// NeuroPLC — Auto-generated IEC 61131-3 SCL
// Graph: mlp | Target: S71200Backend
// Work memory: 75KB | LUT points: 15
// Nodes: 8 | Ops: {'matmul': 4, 'standard_act': 2, 'softmax': 1, 'argmax': 1}


DATA_BLOCK "NeuroPLC_Weights"
{ S7_Optimized_Access := 'FALSE' }
VERSION : 0.1
NON_RETAIN
   STRUCT

   // MatMul 'fc0': W(32×28) + b(32)
   w0 : ARRAY[0..927] OF REAL :=
[0.5694862, -0.0095692, 0.7619486, 0.2215109, -0.3561512, -0.2522623, 0.2582799, 0.0099258
    0.3836571, -0.0658457, 0.1010401, -0.2984352, 0.1934527, -0.2640140, 0.1362384, -0.0190728
    -0.2375232, -0.1084833, -0.3846658, 0.3771667, -0.1136759, -0.1259104, -0.1682155, 0.4097499
    -0.2194012, -0.2356472, -0.1771912, 0.1675407, 0.1454716, -0.3696787, -0.2783369, -0.1873165
    0.0781848, -0.3527579, -0.2131715, -0.4139680, -0.5927966, 0.3198802, -0.5640871, -0.2003005
    0.1832723, 0.2237836, 0.1929916, 0.2185234, 0.1214973, 0.0208249, 0.2776418, 0.6831574
    -0.1655439, -0.2658227, -0.2709237, 0.0986710, 0.1128972, -0.2047481, -0.3872808, 0.1596099
    -0.2523361, 0.2758174, 0.2686562, -0.5177624, -0.1129441, -0.2192100, 0.3343761, -0.0422801
    -0.3068857, 0.2210509, -0.5496964, 0.3709493, 0.0747587, -0.1170707, -0.3195110, 0.0277475
    -0.2577946, 0.0641775, 0.2055912, 0.6039576, -0.5010191, 0.0377836, 0.2038942, -0.0376425
    0.1546009, 0.3260912, -0.1506072, 0.0569262, -0.1928782, -0.1984540, -0.0539345, 0.3094364
    0.2289592, -0.4250050, -0.0399776, 0.0658291, 0.2534966, -0.0973715, -0.3647969, -0.0156060
    -0.5209337, 0.2564455, 0.1338747, 0.3502659, -0.3756513, 0.2530890, 0.0984663, 0.6602526
    0.3365156, -0.2521311, 0.0946512, -0.6085349, -0.5372492, 0.0455726, -0.0786947, 0.0370381
    -0.5858350, -0.7779619, -0.7385424, -0.2071060, 0.2831336, 0.3243212, 0.2366221, -0.2105746
    -0.3834608, -0.6828474, 0.1007835, 0.0381121, 0.3126857, 0.0975034, 0.0499541, -0.0530838
    0.0799674, -0.1505451, -0.4892448, -0.3954702, 0.1594549, 0.2307071, -0.0041823, 0.5944483
    -0.2759206, -0.4257804, -0.3279784, -0.2977980, 0.0038754, 0.3761657, 0.4177073, 0.0741864
    0.3750937, 0.2039272, -0.2429399, -0.3849822, 0.1600508, -0.1581226, -0.0233814, -0.1151747
    -0.5731639, -0.0274457, 0.1195597, -0.2395748, 0.2293357, -0.0251415, 0.3937997, -0.1454628
    -0.0673693, 0.2948158, 0.5630679, -0.3092144, 0.1832785, 0.0043120, 0.0011036, 0.2549984
    0.1242365, -0.1573328, 0.1472307, 0.2971004, 0.1052006, 0.3616425, -0.1347494, -0.3794992
    0.5467421, -0.1476457, 0.3496484, -0.0583753, 0.2853532, -0.3058073, -0.1615329, -0.5229150
    0.2140338, -0.2294949, 0.2921923, 0.0373898, 0.3493846, 0.5938788, 0.0955027, -0.1719695
    0.6582399, -0.4911650, 0.1269870, -0.4129370, -0.2735490, -0.2155660, 0.4269275, -0.1273027
    -0.2414422, -0.3611139, 0.6480063, 0.3808921, -0.2189153, 0.0094489, 0.6784652, 0.3757944
    0.5965886, 0.3704935, 0.3205929, 0.2190031, -0.3913886, 0.2046225, 0.7660633, 0.5648795
    0.0447379, -0.1363681, -0.1653181, -0.3211187, 0.0557173, -0.6775630, 0.2077208, 0.1863764
    0.0122372, -0.1510706, -0.0393031, -0.2373850, 0.3297745, -0.3327326, -0.1183226, 0.3871697
    -0.4481050, -0.2065133, 0.1012533, -0.2578072, 0.0634624, -0.1246978, 0.1465549, -0.5023389
    0.0640146, 0.1963426, 0.6648222, -0.6102669, -0.2871900, -0.3684005, -0.4533643, -0.1819637
    -0.3802012, 0.4682154, 0.1991423, 0.5698866, 0.3063245, 0.1672625, 0.2611240, -0.6845852
    -0.1005014, -0.6641653, -0.2544510, 0.1954752, -0.2994281, 0.3571715, -0.0372742, -0.0310561
    0.1959654, -0.1060541, 0.3827632, -0.3923316, -0.5924090, 0.0670658, 0.3532278, 0.6439264
    0.1193878, -0.5490641, -0.6517076, 0.2266813, 0.2735080, 0.2562127, 0.3711089, -0.0201157
    0.5907255, 0.3026478, 0.0879490, -0.1103418, 0.0830003, 0.0901832, 0.4872787, -0.4248994
    0.6916616, 0.0068263, 0.0377772, -0.3450460, 0.5848706, -0.0756037, 0.0390328, -0.4139087
    -0.1527735, -0.2285863, 0.3310088, 0.2031009, -0.5309294, -0.4607368, 0.1824918, -0.1911459
    -0.1732452, -0.3283744, -0.0425148, -0.0754750, -0.0751830, -0.0057766, -0.0669558, -0.0518108
    -0.1100485, 0.4202482, 0.1722786, 0.2540640, -0.2125306, -0.3108644, -0.1653187, 0.0082027
    0.1613134, 0.5696448, 0.4734836, -0.1820288, -0.0202256, 0.2319008, 0.6178575, -0.1729726
    -0.5705087, -0.4175466, -0.0846097, -0.4305633, -0.0297265, -0.2146564, -0.0228577, 0.4386194
    0.1366172, 0.1275948, 0.2872518, -0.0469490, -0.3430789, -0.2333279, -0.0942715, -0.6695372
    0.3036573, 0.6706407, 0.4867018, 0.2229243, 0.1479198, 0.4786703, -0.1235309, -0.1444162
    -0.1594525, 0.0118241, 0.3302614, 0.4612524, -0.1728074, -0.4940682, 0.2663130, 0.4213447
    0.1559720, 0.0927116, 0.2581408, 0.1484697, 0.5596921, 0.6450443, 0.2316463, -0.3064318
    0.3154030, 0.2504337, 0.2270162, -0.2362736, -0.1822204, 0.7585521, 0.2454521, -0.3572387
    0.1800293, 0.1965537, 0.1946464, 0.1738928, -0.1159788, -0.1791228, 0.3109314, 0.1039406
    -0.2558490, -0.4132357, -0.1826324, -0.0949509, 0.0754630, -0.4951166, -0.0366096, -0.5241205
    0.0701182, 0.5458165, -0.3082272, -0.1620290, 0.2685293, -0.1115321, 0.5528188, 0.1818966
    -0.2705870, -0.4477837, -0.3260813, -0.1751753, 0.3439055, 0.3690660, -0.0775537, -0.3291571
    0.3966570, 0.3747428, 0.2037812, 0.5063270, -0.0363616, -0.0945516, -0.2667596, -0.1880456
    0.2148547, -0.6592890, -0.2238534, -0.2862469, -0.8308039, -0.4430834, -0.0302747, 0.0918460
    -0.3334551, -0.1804388, -0.1097601, 0.3427432, 0.0736062, -0.6790179, -0.2430520, -0.2084594
    0.1491454, -0.0083196, 0.2553293, 0.1678275, 0.0936099, 0.1736043, -0.5376837, -0.4510113
    -0.3174161, 0.2371299, 0.3883051, 0.3464468, 0.1098732, 0.0205052, -0.2641115, -0.3012585
    -0.5463231, -0.0684724, -0.1422806, -0.2644515, -0.4767578, -0.4182616, -0.4673964, -0.0129319
    -0.5374129, -0.1050398, 0.0632549, 0.0568505, 0.2111508, 0.3917949, -0.0330271, 0.2814879
    -0.3214771, 0.3430510, -0.3870021, -0.4042188, 0.1747253, 0.3262924, 0.5594077, 0.0277393
    -0.2604083, 0.0503597, 0.3725081, -0.0544451, 0.0951887, -0.5271522, -0.3720489, 0.0333015
    0.3407656, -0.0524092, -0.3947720, 0.0632993, -0.4918242, -0.0408889, 0.5603451, 0.3429145
    -0.0672607, -0.3218429, -0.3621323, -0.5524946, 0.3105496, 0.3352183, -0.6259544, -0.1107638
    0.0901521, 0.0038500, 0.5420415, 0.2380718, -0.0511688, -0.0771460, -0.0791493, -0.1069665
    0.6399192, -0.0014034, 0.3290343, -0.3565734, 0.2305476, -0.0417552, 0.2942790, -0.1355964
    0.0557771, 0.3271682, -0.3025698, 0.2897500, 0.1278277, -0.1560617, 0.2582703, -0.0549245
    -0.0921321, 0.4996554, 0.0836308, 0.2032579, -0.1741465, -0.2436171, -0.3661414, -0.2924559
    -0.4407195, 0.2304931, -0.2509898, -0.6881460, 0.1500384, 0.4429501, 0.5444623, 0.0644146
    0.1564979, 0.1936211, -0.2217757, 0.1632960, 0.0949209, 0.5449093, 0.3260632, 0.4177442
    -0.1678705, -0.4614883, -0.1780888, 0.0282706, -0.3548764, 0.1119965, -0.6278588, -0.2857478
    0.3291071, -0.2958602, -0.2171935, 0.0488607, -0.2721503, -0.0109805, -0.2872001, -0.3800366
    0.7377275, 0.5175216, 0.4534726, 0.2131705, 0.1694544, 0.1088488, 0.2956495, -0.1219863
    0.4281839, 0.0482728, 0.3261450, 0.0147065, 0.0197347, -0.2837075, -0.2223815, -0.3011971
    0.4010099, 0.3606303, 0.5675586, -0.1933776, 0.1411208, 0.4412328, -0.3157989, 0.0737199
    0.2547267, -0.4104514, 0.3333948, 0.0244799, 0.3485871, -0.1856655, -0.2338329, -0.2214157
    0.4647014, -0.3053385, -0.1758788, -0.2062785, 0.4421045, 0.2903270, 0.2819436, -0.3433319
    -0.0214767, 0.5416198, -0.0143610, -0.1832658, -0.5633022, -0.1308155, 0.1253684, -0.3460040
    -0.0773746, -0.0179889, -0.3036036, 0.0990553, -0.2073587, 0.0275394, 0.0471204, -0.0187443
    0.4038751, 0.0922068, -0.2135524, -0.4082574, -0.0358560, -0.1610684, -0.4163499, 0.2467240
    0.0747931, 0.3987921, 0.1632655, -0.3848493, 0.1649167, -0.6442378, -0.4510081, -0.2822698
    0.4664556, -0.2991767, -0.0362801, -0.3327457, -0.3074295, 0.1606831, -0.0541677, -0.5748461
    0.3949239, -0.2336025, -0.0525538, 0.3131756, -0.0032524, -0.0003879, 0.3644529, 0.3278647
    -0.0496909, -0.0200011, 0.4739185, -0.3886660, 0.0855980, -0.4665208, 0.4008028, -0.5448800
    -0.4093939, -0.1329360, 0.2988919, -0.0788539, 0.0282110, -0.1015701, 0.5736219, -0.2615215
    0.0237927, 0.0321014, -0.1239056, -0.2004481, -0.0194097, -0.1323835, -0.0777957, 0.0366594
    0.1079154, 0.4157223, -0.2902254, 0.4283061, 0.0650300, 0.1249261, -0.2917063, -0.1270394
    0.0782463, 0.5982807, 0.1017760, 0.1843081, -0.6125457, 0.2722199, -0.0728571, -0.5004624
    0.4432183, 0.4912130, 0.0002442, -0.0942999, 0.5940161, -0.1235101, 0.3478113, 0.0345737
    -0.0406947, 0.6151400, 0.2030335, -0.3236780, -0.6019017, -0.4779230, -0.8101817, -0.2094196
    -0.3149875, 0.3055148, -0.2818980, 0.2800311, -0.8234739, -0.6584272, 0.2585062, 0.0584044
    -0.5591815, -0.0547792, 0.0355113, 0.2701355, -0.5936313, 0.3193162, 0.1195579, 0.0537417
    0.6140408, 0.5008627, -0.0104372, 0.2329175, -0.0168664, 0.0332739, 0.3730388, 0.1635417
    0.7335413, 0.5691491, 0.0170918, 0.2825087, 0.0198349, 0.4498756, 0.4100120, -0.2479021
    0.2850291, -0.1702987, -0.4980538, -0.0941117, 0.4272463, -0.2824812, 0.6535753, 0.2375765
    0.4509313, -0.0013205, 0.1127060, -0.1239916, 0.3028973, 0.0927592, -0.3168923, 0.1611173
    0.4917028, 0.0417323, 0.3917417, -0.0557213, -0.2345485, 0.3833969, 0.3747815, -0.1519468
    -0.3892233, -0.0699942, -0.3351573, -0.3026012, -0.1781991, 0.4689204, -0.1804391, -0.2284776
    -0.3932275, 0.2445571, -0.1087966, -0.2825441, -0.2301650, 0.5091258, -0.7006359, 0.0339814
    0.1417895, 0.1839303, 0.2910166, 0.1044962, 0.0580844, 0.6158280, -0.0284938, 0.0542879
    0.1680317, 0.2264472, -0.2030084, 0.0756811, -0.2188872, -0.2264328, -0.1813061, -0.2645762
    0.4621922, -0.4514092, 0.3058094, 0.3434274, 0.3808913, -0.3231871, 0.2469297, -0.1890893
    0.0499585, -0.3218643, 0.6025205, 0.0650566, -0.2298092, 0.5071256, -0.2657916, -0.1830709
    0.0415640, -0.1594847, -0.0321660, -0.0346579, -0.3819390, 0.2074234, 0.3919429, 0.0324158
    -0.0215873, -0.1329270, 0.0735578, 0.3148956, -0.4435450, -0.3320747, -0.1767979, -0.4104172
    0.3253109, -0.1773608, -0.4930988, 0.3281353, 0.3916833, -0.1541856, 0.1263307, 0.0426248
    -0.5533415, 0.0726361, -0.4881184, -0.1073755, -0.5946367, -0.5742470, 0.1233901, -0.0872265
    0.2010813, 0.4012275, 0.3290967, 0.3005436, -0.0111396, -0.4794478, -0.0532993, -0.1733176
    -0.1260332, 0.1089438, 0.0391418, -0.2468968, 0.4689822, -0.4640872, 0.2532913, -0.2343228
    0.2661497, -0.4386278, 0.0468966, -0.3265733, -0.1916417, 0.5178355, 0.2822486, -0.1077720
    0.3286300, -0.0029810, -0.3535745, -0.1011055, 0.1318278, 0.0674391, 0.0591611, -0.1122496
    0.4686061, -0.4002847, 0.0749937, -0.1933431, 0.2702274, -0.1278288, -0.1761822, -0.2737747
    0.4466998, 0.0271071, 0.1916832, 0.4834492, 0.0259246, -0.4892190, 0.2059345, -0.0822330
    -0.4142632, 0.5404200, -0.1093403, 0.0186543, 0.6250578, -0.2241697, 0.3088920, 0.1112378
    -0.1609981, -0.0371174, 0.0221225, 0.0337845, 0.2616802, 0.1264098, 0.1833381, 0.1271529
    0.0488858, 0.0241906, -0.3121075, 0.0973287, -0.0882614, -0.3344531, -0.1306882, 0.1518650
    0.0104939, -0.0685202, -0.0953050, 0.0008646, 0.2513834, 0.0002911, 0.1923783, 0.1726166
    0.3154603, 0.0885571, 0.0390019, 0.0755870, 0.1380671, 0.1447226, 0.0485010, 0.1450995];

   // MatMul 'fc1': W(16×32) + b(16)
   w1 : ARRAY[0..527] OF REAL :=
[0.3448875, -0.0985299, -0.2385274, 0.1068773, 0.5171419, -0.1054032, 0.2936411, -0.4853331
    -0.3005029, 0.2366145, 0.3783182, 0.1278910, 0.0211917, -0.1069832, -0.2683547, -0.0976455
    0.6765909, 0.5036446, 0.3599868, 0.0810751, -0.0792580, -0.2718676, -0.4316851, -0.1867653
    0.2037492, -0.0189868, -0.0119788, 0.3331117, -0.1736732, -0.4839838, -0.0297980, -0.6352752
    0.4027197, -0.5263022, 0.2703936, 0.1180763, -0.3752257, -0.6156019, -0.4087748, 0.1517635
    0.2814839, -0.3188637, 0.4876765, 0.1747880, -0.1799005, -0.3207765, 0.6545156, -0.3893254
    -0.3369366, -0.4376430, 0.0413780, -0.1731163, 0.3791941, 0.0461393, 0.0816816, 0.3956819
    -0.3843228, -0.7061806, -0.6190179, -0.4308152, 0.2132129, 0.4490756, -0.2397823, 0.3091693
    -0.1736172, -0.6044765, 0.2081352, 0.4768652, -0.2759739, 0.1133698, -0.0100859, -0.6772556
    0.5169631, 0.1017481, -0.0672581, -0.4697476, -0.1098660, -0.1401970, -0.4618214, -0.2387714
    -0.3492894, -0.2289385, 0.3859353, 0.3484918, 0.0570800, 0.4838708, 0.4412340, 0.1156965
    0.4213234, -0.2558614, 0.2997079, -0.0041088, -0.2610477, -0.2681805, 0.7025032, 0.4033620
    0.0018223, 0.3965206, -0.1132530, 0.3405365, 0.4333419, 0.0468351, -0.4313038, -0.5938676
    -0.1057017, 0.3874305, -0.3047897, -0.3605830, -0.0865778, 0.0169620, -0.2818013, -0.2056310
    0.2889744, -0.2389124, -0.5219849, -0.5379763, -0.3595321, 0.2131797, 0.2746126, 0.2555465
    -0.3816569, -0.1742714, -0.3458711, -0.4732965, 0.3816739, 0.4522255, 0.4340182, 0.1317699
    0.0887004, -0.1704083, 0.2312619, -0.1512796, 0.1522121, -0.3580639, 0.3120518, -0.0891345
    -0.5189782, 0.6759704, 0.8410841, -0.4388631, 0.3120123, 0.0530660, -0.1540236, -0.1420563
    0.3882907, 0.3881267, 0.4476533, 0.4830106, 0.2335594, 0.1241002, -0.2032309, -0.5769788
    0.3601961, 0.5940281, -0.3626602, 0.1981693, -0.0685700, -0.0704796, 0.0195035, -0.4674689
    -0.2348353, -0.3250483, 0.1978887, -0.0533809, 0.5541837, 0.0647560, 0.1574209, -0.4176951
    -0.0328900, -0.4697271, -0.0496295, -0.1912494, -0.2456453, -0.3518490, 0.0067706, 0.6691334
    0.5995317, 0.3372136, -0.2781896, 0.2096184, -0.4983254, -0.0787928, -0.2063265, -0.2567849
    -0.2985751, 0.2627156, 0.1459312, 0.4578165, 0.0136775, 0.4329558, -0.2819005, 0.0772760
    0.1485205, 0.0424627, -0.5533946, -0.3114872, -0.0971009, 0.1043289, -0.0080725, 0.0561389
    0.1712011, -0.2093053, -0.4844932, 0.5200891, -0.4811763, -0.2097965, -0.1644997, 0.0035760
    0.2773729, 0.4809147, -0.3132524, -0.0345517, 0.5111094, 0.1451371, 0.0575851, 0.1672285
    0.3724994, 0.0500904, -0.0895519, 0.0279228, -0.0756062, -0.6023685, 0.5966649, -0.4288191
    -0.2491551, 0.1842164, 0.1995990, 0.3348442, -0.6874152, 0.0923893, 0.5566139, 0.6076588
    0.4055642, 0.1035502, -0.2282035, 0.0315236, 0.3474000, 0.1027276, 0.0550077, -0.1958367
    -0.1637788, 0.2277053, -0.1716563, 0.1922517, 0.2188656, 0.0905953, -0.2237651, 0.4562837
    -0.4297628, 0.0540233, -0.2155596, -0.4905677, 0.2578664, -0.0752592, 0.3203000, 0.2922962
    0.6623323, -0.2237271, -0.3789170, -0.3014932, 0.3499548, -0.3618023, -0.1381309, -0.2487616
    -0.2042618, -0.3798007, 0.2168026, -0.5617495, 0.5470159, 0.3855161, -0.1744407, -0.0063227
    -0.0175713, 0.4657946, 0.2311470, 0.2995405, -0.2337339, 0.2714463, -0.1801859, -0.2387183
    0.2680195, 0.4208193, 0.0763752, -0.0259924, -0.5796329, -0.4459113, -0.0650182, 0.0992380
    -0.2287219, 0.1592736, 0.2655782, -0.7133095, -0.0750051, 0.1930008, 0.2515846, -0.1046810
    0.3638516, -0.5185701, -0.1378490, 0.1176404, -0.1728815, -0.4648141, -0.0106897, 0.2669196
    -0.2057847, -0.0459625, -0.0872513, -0.5442434, 0.4806913, -0.2794292, 0.6181495, 0.4071167
    -0.3071254, 0.1203253, 0.3505305, -0.5886531, -0.2951987, 0.3731146, 0.2878209, 0.2473200
    -0.1784255, 0.4152616, 0.5053530, 0.2126275, 0.3228098, -0.3918779, -0.1658438, 0.5003296
    -0.0053924, 0.0667791, 0.4097935, 0.1006095, 0.6046916, -0.0676274, -0.1915504, 0.3883604
    0.4911340, 0.5468511, -0.1983627, -0.0676885, -0.3710055, 0.1606412, 0.4564988, -0.5501073
    -0.1039538, -0.0296496, -0.5341417, -0.2000433, 0.2511403, 0.3043574, -0.1509714, 0.4652316
    0.5162573, -0.4559039, 0.1557730, -0.3858083, 0.0727105, -0.4605626, -0.0643399, -0.2012528
    -0.2376907, 0.6337410, 0.7189264, 0.2091954, 0.7626936, 0.3527288, -0.1358239, 0.3472250
    -0.0854939, 0.3039412, 0.2409862, 0.4435183, 0.4328762, -0.0231600, -0.1171540, 0.0108573
    -0.0911193, -0.5950353, -0.1391228, 0.1307337, -0.1149503, -0.0330209, -0.4081971, -0.3619282
    -0.1067709, -0.0438268, 0.1861137, 0.1071503, -0.6722144, 0.5858943, 0.1327110, 0.3459137
    0.3487434, 0.0373104, -0.2565190, 0.4223759, -0.2403768, -0.0137525, 0.1307058, -0.5750338
    -0.6017820, 0.1216069, -0.0930582, 0.0528917, 0.2642088, 0.1213500, -0.0773624, 0.1509228
    0.1637788, -0.0275139, 0.5865979, -0.2206961, 0.5099282, 0.2631257, 0.4237445, 0.4448525
    0.4446503, 0.0053865, -0.5579309, -0.1395655, -0.1579983, -0.3564516, 0.0891758, 0.1217025
    -0.3250042, -0.0731721, 0.5731527, 0.3349074, -0.2764013, 0.3669565, 0.1658501, -0.0952915
    0.1848216, -0.3777516, 0.4125981, -0.2243889, 0.2011978, 0.3032005, 0.0724154, 0.2386405
    -0.4659944, -0.5817581, -0.3680228, -0.5429725, -0.4282436, -0.0057439, 0.1407171, -0.0961595
    -0.0304086, -0.5598830, -0.5288109, 0.2501028, -0.1907448, 0.3364898, 0.3753116, -0.1153062
    -0.0149126, -0.3870158, -0.1154010, 0.0744122, -0.4487402, -0.2563244, 0.0335258, -0.1682583
    0.0443628, 0.3070406, -0.0503107, 0.0992935, 0.5251856, 0.6111719, 0.6419194, 0.1297791
    0.1860752, -0.1274762, 0.3434472, 0.5505610, 0.3397494, -0.5685602, 0.0005795, -0.1080624
    0.3114881, 0.4475129, 0.1615055, -0.4390773, -0.0133804, -0.3265319, -0.5983120, -0.2533576
    0.2004646, -0.2516977, -0.2211783, -0.0643062, 0.1233937, 0.1260124, -0.2689813, 0.3791626
    0.3063162, -0.2886556, -0.1805890, -0.1727612, -0.2364416, -0.0335479, 0.1661869, 0.1447821
    -0.1905543, -0.4342808, -0.0012427, -0.4948293, 0.0922625, 0.0781584, 0.4070034, 0.0575855
    -0.0313972, -0.1867536, 0.2673712, 0.0710777, -0.2155338, 0.0103840, 0.4061291, -0.0612305
    0.0899094, 0.1921517, 0.1069144, -0.0515455, 0.1089574, -0.1325741, 0.2726102, 0.1574048];

   // MatMul 'fc2': W(4×16) + b(4)
   w2 : ARRAY[0..67] OF REAL :=
[-0.0865753, -0.5062438, 0.1554476, 0.7071172, -0.1023560, 0.5811852, -0.6674285, -0.6164539
    -0.8109480, 0.6379222, 0.3449526, -0.0613255, -0.0052660, -0.7050505, -0.6678494, 0.7979829
    -0.0429653, -0.3721911, 0.9616893, -0.2787606, -0.1421925, -0.1321686, 0.1806948, -0.1417111
    -0.4919258, 0.7062184, -0.4885310, -0.5391713, 0.7159519, -0.5416421, 0.8190475, -0.2587632
    0.7209747, -0.5606546, 0.2996863, -0.4360698, 0.6557293, 0.7114502, -0.0711865, -0.5944882
    0.5009670, -0.2733661, 0.0057439, 0.7727029, -0.5340657, 0.0551448, 0.2726173, -0.4893947
    0.2866370, 0.6904863, -0.7133542, 0.1576146, 0.5721015, 0.0582882, -0.7719719, 0.2141585
    -0.2926230, -0.4390040, 0.2077623, 0.5338089, 0.5839869, 0.7652564, -0.3743652, -0.1907377
    -0.1430807, 0.2929625, 0.1342851, -0.1236853];

   // Total: 3 array blocks
   END_STRUCT;
BEGIN
END_DATA_BLOCK

FUNCTION_BLOCK "NeuroPLC_Inference"
{ S7_Optimized_Access := 'FALSE' }
VERSION : 0.1
VAR_INPUT
    features : ARRAY[0..27] OF REAL;
END_VAR

VAR_OUTPUT
    fault_class : INT;
    confidence : REAL;
END_VAR

VAR
    i, j, k : INT;
    sum_val, max_val, t_val : REAL;
    v0 : ARRAY[0..27] OF REAL;
    v1 : ARRAY[0..31] OF REAL;
    v2 : ARRAY[0..31] OF REAL;
    v3 : ARRAY[0..15] OF REAL;
    v4 : ARRAY[0..15] OF REAL;
    v5 : ARRAY[0..3] OF REAL;
    v6 : ARRAY[0..3] OF REAL;
END_VAR

BEGIN
    // ---- Input ----
    FOR i := 0 TO 27 DO
        v0[i] := features[i];
    END_FOR;

    // ---- fc0: MatMul(28→32) ----
    // W = "NeuroPLC_Weights".w0[:896],   b = w0[896:]
    v1[0] := "NeuroPLC_Weights".w0[896 + 0];
    FOR i := 0 TO 27 DO
        v1[0] := v1[0] + "NeuroPLC_Weights".w0[0 + i] * v0[i];
    END_FOR;
    v1[1] := "NeuroPLC_Weights".w0[896 + 1];
    FOR i := 0 TO 27 DO
        v1[1] := v1[1] + "NeuroPLC_Weights".w0[28 + i] * v0[i];
    END_FOR;
    v1[2] := "NeuroPLC_Weights".w0[896 + 2];
    FOR i := 0 TO 27 DO
        v1[2] := v1[2] + "NeuroPLC_Weights".w0[56 + i] * v0[i];
    END_FOR;
    v1[3] := "NeuroPLC_Weights".w0[896 + 3];
    FOR i := 0 TO 27 DO
        v1[3] := v1[3] + "NeuroPLC_Weights".w0[84 + i] * v0[i];
    END_FOR;
    v1[4] := "NeuroPLC_Weights".w0[896 + 4];
    FOR i := 0 TO 27 DO
        v1[4] := v1[4] + "NeuroPLC_Weights".w0[112 + i] * v0[i];
    END_FOR;
    v1[5] := "NeuroPLC_Weights".w0[896 + 5];
    FOR i := 0 TO 27 DO
        v1[5] := v1[5] + "NeuroPLC_Weights".w0[140 + i] * v0[i];
    END_FOR;
    v1[6] := "NeuroPLC_Weights".w0[896 + 6];
    FOR i := 0 TO 27 DO
        v1[6] := v1[6] + "NeuroPLC_Weights".w0[168 + i] * v0[i];
    END_FOR;
    v1[7] := "NeuroPLC_Weights".w0[896 + 7];
    FOR i := 0 TO 27 DO
        v1[7] := v1[7] + "NeuroPLC_Weights".w0[196 + i] * v0[i];
    END_FOR;
    v1[8] := "NeuroPLC_Weights".w0[896 + 8];
    FOR i := 0 TO 27 DO
        v1[8] := v1[8] + "NeuroPLC_Weights".w0[224 + i] * v0[i];
    END_FOR;
    v1[9] := "NeuroPLC_Weights".w0[896 + 9];
    FOR i := 0 TO 27 DO
        v1[9] := v1[9] + "NeuroPLC_Weights".w0[252 + i] * v0[i];
    END_FOR;
    v1[10] := "NeuroPLC_Weights".w0[896 + 10];
    FOR i := 0 TO 27 DO
        v1[10] := v1[10] + "NeuroPLC_Weights".w0[280 + i] * v0[i];
    END_FOR;
    v1[11] := "NeuroPLC_Weights".w0[896 + 11];
    FOR i := 0 TO 27 DO
        v1[11] := v1[11] + "NeuroPLC_Weights".w0[308 + i] * v0[i];
    END_FOR;
    v1[12] := "NeuroPLC_Weights".w0[896 + 12];
    FOR i := 0 TO 27 DO
        v1[12] := v1[12] + "NeuroPLC_Weights".w0[336 + i] * v0[i];
    END_FOR;
    v1[13] := "NeuroPLC_Weights".w0[896 + 13];
    FOR i := 0 TO 27 DO
        v1[13] := v1[13] + "NeuroPLC_Weights".w0[364 + i] * v0[i];
    END_FOR;
    v1[14] := "NeuroPLC_Weights".w0[896 + 14];
    FOR i := 0 TO 27 DO
        v1[14] := v1[14] + "NeuroPLC_Weights".w0[392 + i] * v0[i];
    END_FOR;
    v1[15] := "NeuroPLC_Weights".w0[896 + 15];
    FOR i := 0 TO 27 DO
        v1[15] := v1[15] + "NeuroPLC_Weights".w0[420 + i] * v0[i];
    END_FOR;
    v1[16] := "NeuroPLC_Weights".w0[896 + 16];
    FOR i := 0 TO 27 DO
        v1[16] := v1[16] + "NeuroPLC_Weights".w0[448 + i] * v0[i];
    END_FOR;
    v1[17] := "NeuroPLC_Weights".w0[896 + 17];
    FOR i := 0 TO 27 DO
        v1[17] := v1[17] + "NeuroPLC_Weights".w0[476 + i] * v0[i];
    END_FOR;
    v1[18] := "NeuroPLC_Weights".w0[896 + 18];
    FOR i := 0 TO 27 DO
        v1[18] := v1[18] + "NeuroPLC_Weights".w0[504 + i] * v0[i];
    END_FOR;
    v1[19] := "NeuroPLC_Weights".w0[896 + 19];
    FOR i := 0 TO 27 DO
        v1[19] := v1[19] + "NeuroPLC_Weights".w0[532 + i] * v0[i];
    END_FOR;
    v1[20] := "NeuroPLC_Weights".w0[896 + 20];
    FOR i := 0 TO 27 DO
        v1[20] := v1[20] + "NeuroPLC_Weights".w0[560 + i] * v0[i];
    END_FOR;
    v1[21] := "NeuroPLC_Weights".w0[896 + 21];
    FOR i := 0 TO 27 DO
        v1[21] := v1[21] + "NeuroPLC_Weights".w0[588 + i] * v0[i];
    END_FOR;
    v1[22] := "NeuroPLC_Weights".w0[896 + 22];
    FOR i := 0 TO 27 DO
        v1[22] := v1[22] + "NeuroPLC_Weights".w0[616 + i] * v0[i];
    END_FOR;
    v1[23] := "NeuroPLC_Weights".w0[896 + 23];
    FOR i := 0 TO 27 DO
        v1[23] := v1[23] + "NeuroPLC_Weights".w0[644 + i] * v0[i];
    END_FOR;
    v1[24] := "NeuroPLC_Weights".w0[896 + 24];
    FOR i := 0 TO 27 DO
        v1[24] := v1[24] + "NeuroPLC_Weights".w0[672 + i] * v0[i];
    END_FOR;
    v1[25] := "NeuroPLC_Weights".w0[896 + 25];
    FOR i := 0 TO 27 DO
        v1[25] := v1[25] + "NeuroPLC_Weights".w0[700 + i] * v0[i];
    END_FOR;
    v1[26] := "NeuroPLC_Weights".w0[896 + 26];
    FOR i := 0 TO 27 DO
        v1[26] := v1[26] + "NeuroPLC_Weights".w0[728 + i] * v0[i];
    END_FOR;
    v1[27] := "NeuroPLC_Weights".w0[896 + 27];
    FOR i := 0 TO 27 DO
        v1[27] := v1[27] + "NeuroPLC_Weights".w0[756 + i] * v0[i];
    END_FOR;
    v1[28] := "NeuroPLC_Weights".w0[896 + 28];
    FOR i := 0 TO 27 DO
        v1[28] := v1[28] + "NeuroPLC_Weights".w0[784 + i] * v0[i];
    END_FOR;
    v1[29] := "NeuroPLC_Weights".w0[896 + 29];
    FOR i := 0 TO 27 DO
        v1[29] := v1[29] + "NeuroPLC_Weights".w0[812 + i] * v0[i];
    END_FOR;
    v1[30] := "NeuroPLC_Weights".w0[896 + 30];
    FOR i := 0 TO 27 DO
        v1[30] := v1[30] + "NeuroPLC_Weights".w0[840 + i] * v0[i];
    END_FOR;
    v1[31] := "NeuroPLC_Weights".w0[896 + 31];
    FOR i := 0 TO 27 DO
        v1[31] := v1[31] + "NeuroPLC_Weights".w0[868 + i] * v0[i];
    END_FOR;

    // ---- relu0: RELU ----
    IF v1[0] > 0.0 THEN v2[0] := v1[0]; ELSE v2[0] := 0.0; END_IF;
    IF v1[1] > 0.0 THEN v2[1] := v1[1]; ELSE v2[1] := 0.0; END_IF;
    IF v1[2] > 0.0 THEN v2[2] := v1[2]; ELSE v2[2] := 0.0; END_IF;
    IF v1[3] > 0.0 THEN v2[3] := v1[3]; ELSE v2[3] := 0.0; END_IF;
    IF v1[4] > 0.0 THEN v2[4] := v1[4]; ELSE v2[4] := 0.0; END_IF;
    IF v1[5] > 0.0 THEN v2[5] := v1[5]; ELSE v2[5] := 0.0; END_IF;
    IF v1[6] > 0.0 THEN v2[6] := v1[6]; ELSE v2[6] := 0.0; END_IF;
    IF v1[7] > 0.0 THEN v2[7] := v1[7]; ELSE v2[7] := 0.0; END_IF;
    IF v1[8] > 0.0 THEN v2[8] := v1[8]; ELSE v2[8] := 0.0; END_IF;
    IF v1[9] > 0.0 THEN v2[9] := v1[9]; ELSE v2[9] := 0.0; END_IF;
    IF v1[10] > 0.0 THEN v2[10] := v1[10]; ELSE v2[10] := 0.0; END_IF;
    IF v1[11] > 0.0 THEN v2[11] := v1[11]; ELSE v2[11] := 0.0; END_IF;
    IF v1[12] > 0.0 THEN v2[12] := v1[12]; ELSE v2[12] := 0.0; END_IF;
    IF v1[13] > 0.0 THEN v2[13] := v1[13]; ELSE v2[13] := 0.0; END_IF;
    IF v1[14] > 0.0 THEN v2[14] := v1[14]; ELSE v2[14] := 0.0; END_IF;
    IF v1[15] > 0.0 THEN v2[15] := v1[15]; ELSE v2[15] := 0.0; END_IF;
    IF v1[16] > 0.0 THEN v2[16] := v1[16]; ELSE v2[16] := 0.0; END_IF;
    IF v1[17] > 0.0 THEN v2[17] := v1[17]; ELSE v2[17] := 0.0; END_IF;
    IF v1[18] > 0.0 THEN v2[18] := v1[18]; ELSE v2[18] := 0.0; END_IF;
    IF v1[19] > 0.0 THEN v2[19] := v1[19]; ELSE v2[19] := 0.0; END_IF;
    IF v1[20] > 0.0 THEN v2[20] := v1[20]; ELSE v2[20] := 0.0; END_IF;
    IF v1[21] > 0.0 THEN v2[21] := v1[21]; ELSE v2[21] := 0.0; END_IF;
    IF v1[22] > 0.0 THEN v2[22] := v1[22]; ELSE v2[22] := 0.0; END_IF;
    IF v1[23] > 0.0 THEN v2[23] := v1[23]; ELSE v2[23] := 0.0; END_IF;
    IF v1[24] > 0.0 THEN v2[24] := v1[24]; ELSE v2[24] := 0.0; END_IF;
    IF v1[25] > 0.0 THEN v2[25] := v1[25]; ELSE v2[25] := 0.0; END_IF;
    IF v1[26] > 0.0 THEN v2[26] := v1[26]; ELSE v2[26] := 0.0; END_IF;
    IF v1[27] > 0.0 THEN v2[27] := v1[27]; ELSE v2[27] := 0.0; END_IF;
    IF v1[28] > 0.0 THEN v2[28] := v1[28]; ELSE v2[28] := 0.0; END_IF;
    IF v1[29] > 0.0 THEN v2[29] := v1[29]; ELSE v2[29] := 0.0; END_IF;
    IF v1[30] > 0.0 THEN v2[30] := v1[30]; ELSE v2[30] := 0.0; END_IF;
    IF v1[31] > 0.0 THEN v2[31] := v1[31]; ELSE v2[31] := 0.0; END_IF;

    // ---- fc1: MatMul(32→16) ----
    // W = "NeuroPLC_Weights".w1[:512],   b = w1[512:]
    v3[0] := "NeuroPLC_Weights".w1[512 + 0];
    FOR i := 0 TO 31 DO
        v3[0] := v3[0] + "NeuroPLC_Weights".w1[0 + i] * v2[i];
    END_FOR;
    v3[1] := "NeuroPLC_Weights".w1[512 + 1];
    FOR i := 0 TO 31 DO
        v3[1] := v3[1] + "NeuroPLC_Weights".w1[32 + i] * v2[i];
    END_FOR;
    v3[2] := "NeuroPLC_Weights".w1[512 + 2];
    FOR i := 0 TO 31 DO
        v3[2] := v3[2] + "NeuroPLC_Weights".w1[64 + i] * v2[i];
    END_FOR;
    v3[3] := "NeuroPLC_Weights".w1[512 + 3];
    FOR i := 0 TO 31 DO
        v3[3] := v3[3] + "NeuroPLC_Weights".w1[96 + i] * v2[i];
    END_FOR;
    v3[4] := "NeuroPLC_Weights".w1[512 + 4];
    FOR i := 0 TO 31 DO
        v3[4] := v3[4] + "NeuroPLC_Weights".w1[128 + i] * v2[i];
    END_FOR;
    v3[5] := "NeuroPLC_Weights".w1[512 + 5];
    FOR i := 0 TO 31 DO
        v3[5] := v3[5] + "NeuroPLC_Weights".w1[160 + i] * v2[i];
    END_FOR;
    v3[6] := "NeuroPLC_Weights".w1[512 + 6];
    FOR i := 0 TO 31 DO
        v3[6] := v3[6] + "NeuroPLC_Weights".w1[192 + i] * v2[i];
    END_FOR;
    v3[7] := "NeuroPLC_Weights".w1[512 + 7];
    FOR i := 0 TO 31 DO
        v3[7] := v3[7] + "NeuroPLC_Weights".w1[224 + i] * v2[i];
    END_FOR;
    v3[8] := "NeuroPLC_Weights".w1[512 + 8];
    FOR i := 0 TO 31 DO
        v3[8] := v3[8] + "NeuroPLC_Weights".w1[256 + i] * v2[i];
    END_FOR;
    v3[9] := "NeuroPLC_Weights".w1[512 + 9];
    FOR i := 0 TO 31 DO
        v3[9] := v3[9] + "NeuroPLC_Weights".w1[288 + i] * v2[i];
    END_FOR;
    v3[10] := "NeuroPLC_Weights".w1[512 + 10];
    FOR i := 0 TO 31 DO
        v3[10] := v3[10] + "NeuroPLC_Weights".w1[320 + i] * v2[i];
    END_FOR;
    v3[11] := "NeuroPLC_Weights".w1[512 + 11];
    FOR i := 0 TO 31 DO
        v3[11] := v3[11] + "NeuroPLC_Weights".w1[352 + i] * v2[i];
    END_FOR;
    v3[12] := "NeuroPLC_Weights".w1[512 + 12];
    FOR i := 0 TO 31 DO
        v3[12] := v3[12] + "NeuroPLC_Weights".w1[384 + i] * v2[i];
    END_FOR;
    v3[13] := "NeuroPLC_Weights".w1[512 + 13];
    FOR i := 0 TO 31 DO
        v3[13] := v3[13] + "NeuroPLC_Weights".w1[416 + i] * v2[i];
    END_FOR;
    v3[14] := "NeuroPLC_Weights".w1[512 + 14];
    FOR i := 0 TO 31 DO
        v3[14] := v3[14] + "NeuroPLC_Weights".w1[448 + i] * v2[i];
    END_FOR;
    v3[15] := "NeuroPLC_Weights".w1[512 + 15];
    FOR i := 0 TO 31 DO
        v3[15] := v3[15] + "NeuroPLC_Weights".w1[480 + i] * v2[i];
    END_FOR;

    // ---- relu1: RELU ----
    IF v3[0] > 0.0 THEN v4[0] := v3[0]; ELSE v4[0] := 0.0; END_IF;
    IF v3[1] > 0.0 THEN v4[1] := v3[1]; ELSE v4[1] := 0.0; END_IF;
    IF v3[2] > 0.0 THEN v4[2] := v3[2]; ELSE v4[2] := 0.0; END_IF;
    IF v3[3] > 0.0 THEN v4[3] := v3[3]; ELSE v4[3] := 0.0; END_IF;
    IF v3[4] > 0.0 THEN v4[4] := v3[4]; ELSE v4[4] := 0.0; END_IF;
    IF v3[5] > 0.0 THEN v4[5] := v3[5]; ELSE v4[5] := 0.0; END_IF;
    IF v3[6] > 0.0 THEN v4[6] := v3[6]; ELSE v4[6] := 0.0; END_IF;
    IF v3[7] > 0.0 THEN v4[7] := v3[7]; ELSE v4[7] := 0.0; END_IF;
    IF v3[8] > 0.0 THEN v4[8] := v3[8]; ELSE v4[8] := 0.0; END_IF;
    IF v3[9] > 0.0 THEN v4[9] := v3[9]; ELSE v4[9] := 0.0; END_IF;
    IF v3[10] > 0.0 THEN v4[10] := v3[10]; ELSE v4[10] := 0.0; END_IF;
    IF v3[11] > 0.0 THEN v4[11] := v3[11]; ELSE v4[11] := 0.0; END_IF;
    IF v3[12] > 0.0 THEN v4[12] := v3[12]; ELSE v4[12] := 0.0; END_IF;
    IF v3[13] > 0.0 THEN v4[13] := v3[13]; ELSE v4[13] := 0.0; END_IF;
    IF v3[14] > 0.0 THEN v4[14] := v3[14]; ELSE v4[14] := 0.0; END_IF;
    IF v3[15] > 0.0 THEN v4[15] := v3[15]; ELSE v4[15] := 0.0; END_IF;

    // ---- fc2: MatMul(16→4) ----
    // W = "NeuroPLC_Weights".w2[:64],   b = w2[64:]
    v5[0] := "NeuroPLC_Weights".w2[64 + 0];
    FOR i := 0 TO 15 DO
        v5[0] := v5[0] + "NeuroPLC_Weights".w2[0 + i] * v4[i];
    END_FOR;
    v5[1] := "NeuroPLC_Weights".w2[64 + 1];
    FOR i := 0 TO 15 DO
        v5[1] := v5[1] + "NeuroPLC_Weights".w2[16 + i] * v4[i];
    END_FOR;
    v5[2] := "NeuroPLC_Weights".w2[64 + 2];
    FOR i := 0 TO 15 DO
        v5[2] := v5[2] + "NeuroPLC_Weights".w2[32 + i] * v4[i];
    END_FOR;
    v5[3] := "NeuroPLC_Weights".w2[64 + 3];
    FOR i := 0 TO 15 DO
        v5[3] := v5[3] + "NeuroPLC_Weights".w2[48 + i] * v4[i];
    END_FOR;

    // ---- softmax: Softmax ----
    v6[0] := EXP(v5[0]);
    v6[1] := EXP(v5[1]);
    v6[2] := EXP(v5[2]);
    v6[3] := EXP(v5[3]);
    sum_val := v6[0]
             + v6[1]
             + v6[2]
             + v6[3]
             ;
    IF sum_val > 0.0 THEN
        v6[0] := v6[0] / sum_val;
        v6[1] := v6[1] / sum_val;
        v6[2] := v6[2] / sum_val;
        v6[3] := v6[3] / sum_val;
    END_IF;

    // ---- Argmax ----
    max_val := v7[0];
    fault_class := 0;
    IF v7[1] > max_val THEN
        max_val := v7[1];
        fault_class := 1;
    END_IF;
    IF v7[2] > max_val THEN
        max_val := v7[2];
        fault_class := 2;
    END_IF;
    IF v7[3] > max_val THEN
        max_val := v7[3];
        fault_class := 3;
    END_IF;
    confidence := max_val;

END_FUNCTION_BLOCK